PROGRAM MAIN
VAR
END_VAR

END_PROGRAM

(* stored: Version 1.1.0.1
   POU MAIN: Id {e11e88b4-816c-43c1-b5d0-c1882815007f} *)
